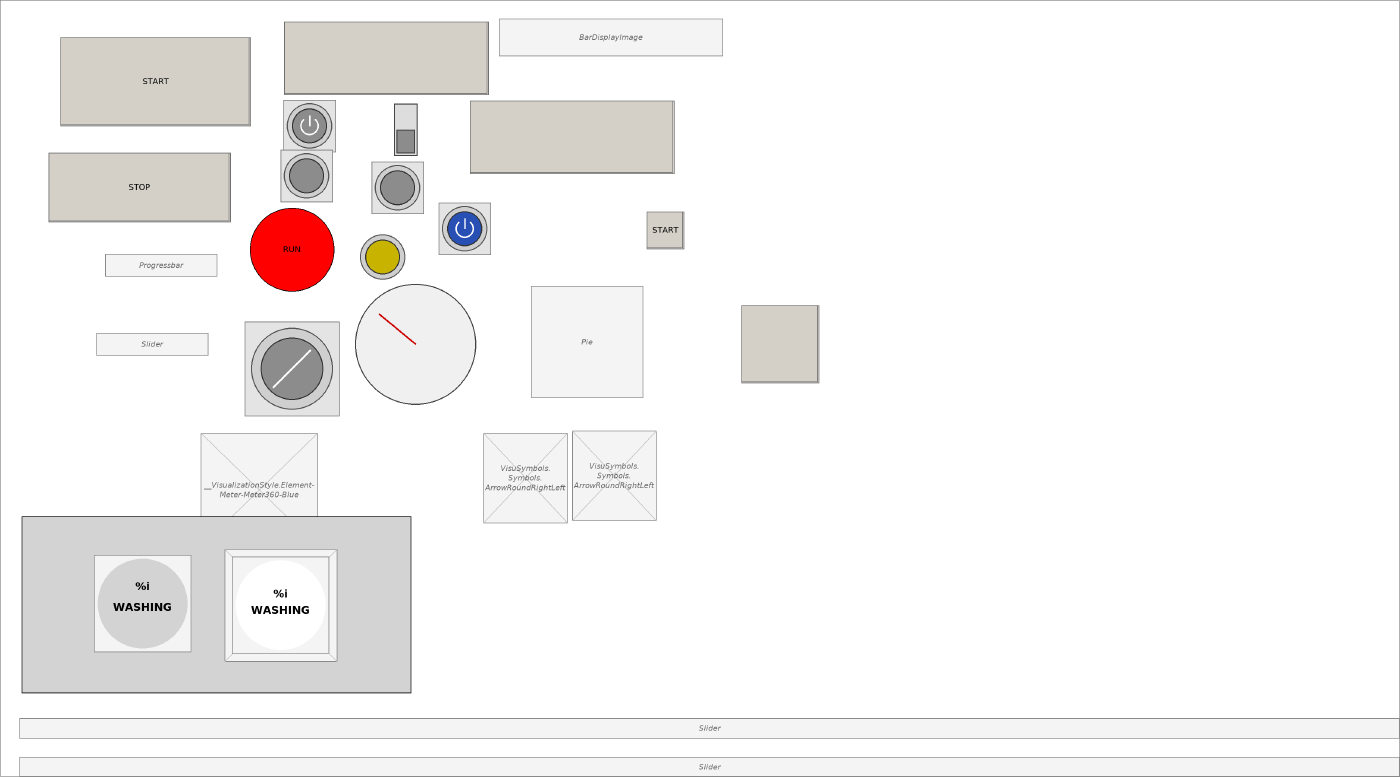
VISUALIZATION Visualization  // 1877x1043
    Button (81,50 255x119), "START"
        tap StartStop.Start
    Button (65,205 244x93), "STOP"
        tap StartStop.Stop
    DipSwitch (509,139 70x70), variable: StartStop.Start, behaviour: TOGGLE, style: Switch-DipSwitch-Gray
    Lamp1 (478,310 70x70), variable: StartStop.Run, style: Lamp-Lamp1-Yellow
    PowerSwitch (380,134 70x70), variable: StartStop.Start, behaviour: TOGGLE, style: Switch-PowerSwitch-Gray
    PushSwitch (376,201 70x70), variable: StartStop.Start, behaviour: TOGGLE, style: Switch-PushSwitch-Gray
    PushSwitchLed (498,217 70x70), variable: StartStop.Start, behaviour: TOGGLE, style: Switch-PushSwitchLed-Gray
    RockerSwitch (476,46 70x70), variable: StartStop.Start, behaviour: TOGGLE, style: Switch-RockerSwitch-Gray
    RotarySwitch (571,43 70x70), variable: StartStop.Start, behaviour: TOGGLE, style: Switch-RotarySwitch-Gray
    BarDisplayImage (669,25 300x50), value: StartStop.Value, style: BarDisplayImage-Gray, scale format: %.1f, scale 0..100
    Meter360 (476,379 162x166), value: StartStop.Value, style: Meter-Meter360-Gray, scale format: %.1f, scale 0..100
    Potentiometer360 (328,427 127x136), variable: StartStop.Value, style: Potentiometer-Potentiometer360-Gray, scale format: %.1f, scale 0..100
        p2431819421: Outside
    Progressbar (141,341 150x30), variable: StartStop.Value
    Slider (129,447 150x30), variable: StartStop.Value, scale 0..100
    Pie (712,384 150x150)
        p426801730: StartStop.Value
    Image (269,581 157x153)
        p573394764: StartStop.Value
    Ellipse (335,279 113x112), "RUN", colour toggle: StartStop.Run
    PowerSwitch (588,272 70x70), variable: StartStop.Start, behaviour: TOGGLE, style: Switch-PowerSwitch-Blue
    Image (648,581 113x121), image: VisuSymbols.Symbols.ArrowRoundRightLeft
        p2277200375: StartStop.Value
    Image (767,578 113x121), image: VisuSymbols.Symbols.ArrowRoundRightLeft
        p2858320360: StartStop.Value
    Button (630,135 274x98)
        OnMouseClick: toggle StartStop.Stop
    Button (381,29 274x98)
        OnMouseClick: change screen: Login_Page
    Button (867,284 50x50), "START", image: VisuSymbols.Symbols.TriangleDown
        tap StartStop.Start
    Rectangle (29,693 522x237)
    Pie (126,745 130x130)
        p426801730: StartStop.Value
        p2124672552: StartStop.FAIZValue2
    Ellipse (131,750 120x120), colour toggle: StartStop.Start
        toggle StartStop.Start
    Label (171,782 40x24)
    Label (150,803 82x24), "WASHING"
    Image (301,737 151x151)
        p573394764: StartStop.Value
    Pie (311,747 130x130)
        p426801730: StartStop.Value
        p2124672552: StartStop.FAIZValue2
    Ellipse (316,752 120x120), colour toggle: StartStop.Start
        toggle StartStop.Start
    Rectangle (342,782 69x30), "%i", text variable: StartStop.Value
    Rectangle (157,772 69x30), "%i", text variable: StartStop.Value
    Label (335,807 82x24), "WASHING"
    Slider (26,964 1851x27), variable: StartStop.Value, scale 0..360
    Slider (26,1016 1851x27), variable: StartStop.FAIZValue2, scale 0..360
    Button (994,410 104x104)
END_VISUALIZATION

(* stored: Version 1.1.0.1, ProductVersion 3.1.4024.12
   Visu Visualization: Id {c022df96-5cc6-4943-9058-f73de1ab6bfa} *)
